DATA_BLOCK "MyCounter_DB0"
{ S7_Optimized_Access := 'TRUE' }
VERSION : 0.1
NON_RETAIN
"MyCounter"

BEGIN

END_DATA_BLOCK

